# EPICS substitutions: gigeApp/Db/iocAdmin.substitutions
#==============================================================================
#
# Abs:  IOC Administration Records
#
# Name: iocAdmin.substitutions
#
#==============================================================================
#
file iocSoft.db
{
	pattern
	{ IOC = '$(IOC)'	}
}
